(* IEC 61131-3 sources: eCockpitGit/test_project/src/%F%00 Library/%F%Common Functions/%F%Buffer/%POU%FB_FIFOQueue/%PRO%isEmpty, 1 file *)

(* ---- %GETSET%Get.st ---- *)
//Returns whether the buffer is empty
// |**Version**|**Author**| **Date** |**Changes**
// | 1         | NSN      | 15-02-22 | Creation
VAR
END_VAR

(*%!%__DELIMITER__%!%*)
isEmpty		:=		S_amount = 0;
